FUNCTION_BLOCK FB_Stop
VAR_INPUT
(*È«¾Ö*)
	Mode:DINT;
	PowerState:DINT;
	CoupleState:DINT;
	(*GapMode*)
	GapStop:BOOL;
	(*BCGapMode*)
	BCGapStop:BOOL;
	(*SingleCarrierMode*)
	TopStop:BOOL;
	BottomStop:BOOL;
	(*TaperMode*)
	TaperStop:BOOL;
	(*DebugMode*)
	LeftTopStop:BOOL;
	RightTopStop:BOOL;
	LeftBottomStop:BOOL;
	RightBottomStop:BOOL;
END_VAR
VAR_OUTPUT
	FbID:DINT:=1001;
	GapState:DINT;
	GapBusy:BOOL;
	GapDone:BOOL;

	BCGapState:DINT;
	BCGapBusy:BOOL;
	BCGapDone:BOOL;

	TopState:DINT;
	TopBusy:BOOL;
	TopDone:BOOL;
	BottomState:DINT;
	BottomBusy:BOOL;
	BottomDone:BOOL;

	TaperState:DINT;
	TaperBusy:BOOL;
	TaperDone:BOOL;

	LeftTopState:DINT;
	LeftTopBusy:BOOL;
	LeftTopDone:BOOL;
	RightTopState:DINT;
	RightTopBusy:BOOL;
	RightTopDone:BOOL;
	LeftBottomState:DINT;
	LeftBottomBusy:BOOL;
	LeftBottomDone:BOOL;
	RightBottomState:DINT;
	RightBottomBusy:BOOL;
	RightBottomDone:BOOL;

	Error:BOOL;
	ErrorID:DINT;
END_VAR
VAR
	Top_MC_Stop: MC_Stop;
	Bottom_MC_Stop: MC_Stop;
	RightTopLin_MC_Stop: MC_Stop;
	RightBottomLin_MC_Stop: MC_Stop;
	fb_ton: TON;
	fb_ton1: TON;
	fb_ton2: TON;
	fb_ton_debug_1:TON;
	fb_ton_debug_2:TON;
	fb_ton_debug_3:TON;
	fb_ton_debug_4:TON;
	fb_ton_BC: TON;
END_VAR

IF PowerState=1 THEN
	IF Mode=1 AND CoupleState=1 THEN
		A_GapStop();
	ELSIF Mode=2 AND CoupleState=1 AND TopStop THEN
		A_TopStop();
	ELSIF Mode=2 AND CoupleState=1 AND BottomStop THEN
		A_BottomStop();
	ELSIF Mode=3 AND CoupleState=0 AND TaperStop THEN
		A_TaperStop();
	ELSIF Mode=4 AND CoupleState=0 AND LeftTopStop THEN
		A_LeftTopStop();
	ELSIF Mode=4 AND CoupleState=0 AND RightTopStop THEN
		A_RightTopStop();
	ELSIF Mode=4 AND CoupleState=0 AND LeftBottomStop THEN
		A_LeftBottomStop();
	ELSIF Mode=4 AND CoupleState=0 AND RightBottomStop THEN
		A_RightBottomStop();
	ELSIF Mode=5 AND CoupleState=0 AND BCGapStop THEN
		A_BCGapStop();
	ELSE
		FB_PlcEmergencyStop();
	END_IF
END_IF

ACTION A_BCGapStop:
IF BCGapStop THEN
BCGapBusy:=TRUE;
BCGapDone:=FALSE;
fb_ton_BC(PT:=t#100ms);
A_StopMC();
CASE BCGapState OF
	0:
		IF Top_MC_Stop.Error OR Bottom_MC_Stop.Error OR RightTopLin_MC_Stop.Error OR RightBottomLin_MC_Stop.Error THEN
			ErrorID:=1;
			BCGapState:=-100;
			Top_MC_Stop.Execute:=FALSE;
			Bottom_MC_Stop.Execute:=FALSE;
			RightTopLin_MC_Stop.Execute:=FALSE;
			RightBottomLin_MC_Stop.Execute:=FALSE;
			A_StopMC();
		ELSE
			BCGapState:=1;
		END_IF
	1:
		Top_MC_Stop.Execute:=TRUE;
		Bottom_MC_Stop.Execute:=TRUE;
		RightTopLin_MC_Stop.Execute:=TRUE;
		RightBottomLin_MC_Stop.Execute:=TRUE;
		fb_ton_BC.IN:=TRUE;
		BCGapState:=2;
	2:
		IF  NOT Top_MC_Stop.Done OR NOT Bottom_MC_Stop.Done OR NOT RightTopLin_MC_Stop.Done OR NOT RightBottomLin_MC_Stop.Done THEN
				BCGapState:=2;
		ELSE
			BCGapState:=88;
			Top_MC_Stop.Execute:=FALSE;
			Bottom_MC_Stop.Execute:=FALSE;
			RightTopLin_MC_Stop.Execute:=FALSE;
			RightBottomLin_MC_Stop.Execute:=FALSE;
			A_StopMC();
		END_IF

	88:
		BCGapStop:=FALSE;
		BCGapState:=0;
		BCGapBusy:=FALSE;
		BCGapDone:=TRUE;
		Error:=FALSE;
		ErrorID:=0;
		fb_ton_BC.IN:=FALSE;

	-100:
		FB_PlcEmergencyStop();
		BCGapStop:=FALSE;
		BCGapState:=-100;
		BCGapBusy:=FALSE;
		BCGapDone:=FALSE;
		Error:=TRUE;
		Top_MC_Stop.Execute:=FALSE;
		Bottom_MC_Stop.Execute:=FALSE;
		RightTopLin_MC_Stop.Execute:=FALSE;
		RightBottomLin_MC_Stop.Execute:=FALSE;
		A_StopMC();
		fb_ton_BC.IN:=FALSE;

END_CASE
END_IF
END_ACTION

ACTION A_BottomStop:
IF BottomStop THEN
BottomBusy:=TRUE;
BottomDone:=FALSE;
fb_ton2(PT:=t#100ms);
A_StopMC();
CASE BottomState OF
	0:
		IF Bottom_MC_Stop.Error THEN
			ErrorID:=1;
			BottomState:=-100;
			Bottom_MC_Stop.Execute:=FALSE;
			A_StopMC();
		ELSE
			BottomState:=1;
		END_IF
	1:
		Bottom_MC_Stop.Execute:=TRUE;
		fb_ton2.IN:=TRUE;
		BottomState:=2;
	2:
		IF  NOT Bottom_MC_Stop.Done THEN
				BottomState:=2;
		ELSE
			BottomState:=88;
			Bottom_MC_Stop.Execute:=FALSE;
			A_StopMC();
		END_IF

	88:
		BottomStop:=FALSE;
		BottomState:=0;
		BottomBusy:=FALSE;
		BottomDone:=TRUE;
		Error:=FALSE;
		ErrorID:=0;
		fb_ton2.IN:=FALSE;

	-100:
		FB_PlcEmergencyStop();
		BottomStop:=FALSE;
		BottomState:=-100;
		BottomBusy:=FALSE;
		BottomDone:=FALSE;
		Error:=TRUE;
		Bottom_MC_Stop.Execute:=FALSE;
		A_StopMC();
		fb_ton2.IN:=FALSE;

END_CASE
END_IF
END_ACTION

ACTION A_GapStop:
IF GapStop THEN
GapBusy:=TRUE;
GapDone:=FALSE;
fb_ton(PT:=t#100ms);
A_StopMC();
CASE GapState OF
	0:
		IF Top_MC_Stop.Error OR Bottom_MC_Stop.Error THEN
			ErrorID:=1;
			GapState:=-100;
			Top_MC_Stop.Execute:=FALSE;
			Bottom_MC_Stop.Execute:=FALSE;
			A_StopMC();
		ELSE
			GapState:=1;
		END_IF
	1:
		Top_MC_Stop.Execute:=TRUE;
		Bottom_MC_Stop.Execute:=TRUE;
		fb_ton.IN:=TRUE;
		GapState:=2;
	2:
		IF  NOT Top_MC_Stop.Done OR NOT Bottom_MC_Stop.Done THEN
				GapState:=2;
		ELSE
			GapState:=88;
			Top_MC_Stop.Execute:=FALSE;
			Bottom_MC_Stop.Execute:=FALSE;
			A_StopMC();
		END_IF

	88:
		GapStop:=FALSE;
		GapState:=0;
		GapBusy:=FALSE;
		GapDone:=TRUE;
		Error:=FALSE;
		ErrorID:=0;
		fb_ton.IN:=FALSE;

	-100:
		FB_PlcEmergencyStop();
		GapStop:=FALSE;
		GapState:=-100;
		GapBusy:=FALSE;
		GapDone:=FALSE;
		Error:=TRUE;
		Top_MC_Stop.Execute:=FALSE;
		Bottom_MC_Stop.Execute:=FALSE;
		A_StopMC();
		fb_ton.IN:=FALSE;

END_CASE
END_IF
END_ACTION

ACTION A_LeftBottomStop:
IF LeftBottomStop THEN
LeftBottomBusy:=TRUE;
LeftBottomDone:=FALSE;
fb_ton_debug_3(PT:=t#100ms);
A_StopMC();
CASE LeftBottomState OF
	0:
		IF Bottom_MC_Stop.Error THEN
			ErrorID:=41;
			LeftBottomState:=-100;
			Bottom_MC_Stop.Execute:=FALSE;
			A_StopMC();
		ELSE
			LeftBottomState:=1;
		END_IF
	1:
		Bottom_MC_Stop.Execute:=TRUE;
		fb_ton_debug_3.IN:=TRUE;
		LeftBottomState:=2;
	2:
		IF  NOT Bottom_MC_Stop.Done THEN
				LeftBottomState:=2;
		ELSE
			LeftBottomState:=88;
			Bottom_MC_Stop.Execute:=FALSE;
			A_StopMC();
		END_IF

	88:
		LeftBottomStop:=FALSE;
		LeftBottomState:=0;
		LeftBottomBusy:=FALSE;
		LeftBottomDone:=TRUE;
		Error:=FALSE;
		ErrorID:=0;
		fb_ton_debug_3.IN:=FALSE;

	-100:
		FB_PlcEmergencyStop();
		LeftBottomStop:=FALSE;
		LeftBottomState:=-100;
		LeftBottomBusy:=FALSE;
		LeftBottomDone:=FALSE;
		Error:=TRUE;
		Bottom_MC_Stop.Execute:=FALSE;
		A_StopMC();
		fb_ton_debug_3.IN:=FALSE;

END_CASE
END_IF
END_ACTION

ACTION A_LeftTopStop:
IF LeftTopStop THEN
LeftTopBusy:=TRUE;
LeftTopDone:=FALSE;
fb_ton_debug_1(PT:=t#100ms);
A_StopMC();
CASE LeftTopState OF
	0:
		IF Top_MC_Stop.Error THEN
			ErrorID:=41;
			LeftTopState:=-100;
			Top_MC_Stop.Execute:=FALSE;
			A_StopMC();
		ELSE
			LeftTopState:=1;
		END_IF
	1:
		Top_MC_Stop.Execute:=TRUE;
		fb_ton_debug_1.IN:=TRUE;
		LeftTopState:=2;
	2:
		IF  NOT Top_MC_Stop.Done THEN
				LeftTopState:=2;
		ELSE
			LeftTopState:=88;
			Top_MC_Stop.Execute:=FALSE;
			A_StopMC();
		END_IF

	88:
		LeftTopStop:=FALSE;
		LeftTopState:=0;
		LeftTopBusy:=FALSE;
		LeftTopDone:=TRUE;
		Error:=FALSE;
		ErrorID:=0;
		fb_ton_debug_1.IN:=FALSE;

	-100:
		FB_PlcEmergencyStop();
		LeftTopStop:=FALSE;
		LeftTopState:=-100;
		LeftTopBusy:=FALSE;
		LeftTopDone:=FALSE;
		Error:=TRUE;
		Top_MC_Stop.Execute:=FALSE;
		A_StopMC();
		fb_ton_debug_1.IN:=FALSE;

END_CASE
END_IF
END_ACTION

ACTION A_RightBottomStop:
IF RightBottomStop THEN
RightBottomBusy:=TRUE;
RightBottomDone:=FALSE;
fb_ton_debug_4(PT:=t#100ms);
A_StopMC();
CASE RightBottomState OF
	0:
		IF RightBottomLin_MC_Stop.Error THEN
			ErrorID:=41;
			RightBottomState:=-100;
			RightBottomLin_MC_Stop.Execute:=FALSE;
			A_StopMC();
		ELSE
			RightBottomState:=1;
		END_IF
	1:
		RightBottomLin_MC_Stop.Execute:=TRUE;
		fb_ton_debug_4.IN:=TRUE;
		RightBottomState:=2;
	2:
		IF  NOT RightBottomLin_MC_Stop.Done THEN
				RightBottomState:=2;
		ELSE
			RightBottomState:=88;
			RightBottomLin_MC_Stop.Execute:=FALSE;
			A_StopMC();
		END_IF

	88:
		RightBottomStop:=FALSE;
		RightBottomState:=0;
		RightBottomBusy:=FALSE;
		RightBottomDone:=TRUE;
		Error:=FALSE;
		ErrorID:=0;
		fb_ton_debug_4.IN:=FALSE;

	-100:
		FB_PlcEmergencyStop();
		RightBottomStop:=FALSE;
		RightBottomState:=-100;
		RightBottomBusy:=FALSE;
		RightBottomDone:=FALSE;
		Error:=TRUE;
		RightBottomLin_MC_Stop.Execute:=FALSE;
		A_StopMC();
		fb_ton_debug_4.IN:=FALSE;

END_CASE
END_IF
END_ACTION

ACTION A_RightTopStop:
IF RightTopStop THEN
RightTopBusy:=TRUE;
RightTopDone:=FALSE;
fb_ton_debug_2(PT:=t#100ms);
A_StopMC();
CASE RightTopState OF
	0:
		IF RightTopLin_MC_Stop.Error THEN
			ErrorID:=41;
			RightTopState:=-100;
			RightTopLin_MC_Stop.Execute:=FALSE;
			A_StopMC();
		ELSE
			RightTopState:=1;
		END_IF
	1:
		RightTopLin_MC_Stop.Execute:=TRUE;
		fb_ton_debug_2.IN:=TRUE;
		RightTopState:=2;
	2:
		IF  NOT RightTopLin_MC_Stop.Done THEN
				RightTopState:=2;
		ELSE
			RightTopState:=88;
			RightTopLin_MC_Stop.Execute:=FALSE;
			A_StopMC();
		END_IF

	88:
		RightTopStop:=FALSE;
		RightTopState:=0;
		RightTopBusy:=FALSE;
		RightTopDone:=TRUE;
		Error:=FALSE;
		ErrorID:=0;
		fb_ton_debug_2.IN:=FALSE;

	-100:
		FB_PlcEmergencyStop();
		RightTopStop:=FALSE;
		RightTopState:=-100;
		RightTopBusy:=FALSE;
		RightTopDone:=FALSE;
		Error:=TRUE;
		RightTopLin_MC_Stop.Execute:=FALSE;
		A_StopMC();
		fb_ton_debug_2.IN:=FALSE;

END_CASE
END_IF
END_ACTION

ACTION A_StopMC:
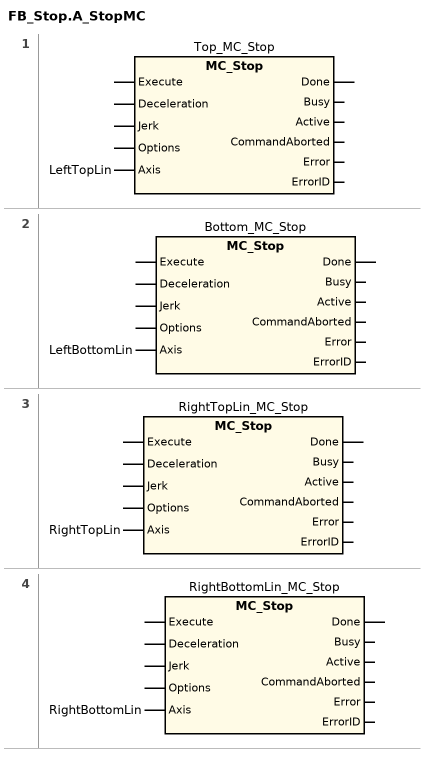
// NETWORK 1
Top_MC_Stop(Axis := LeftTopLin); // MC_Stop

// NETWORK 2
Bottom_MC_Stop(Axis := LeftBottomLin); // MC_Stop

// NETWORK 3
RightTopLin_MC_Stop(Axis := RightTopLin); // MC_Stop

// NETWORK 4
RightBottomLin_MC_Stop(Axis := RightBottomLin); // MC_Stop
END_ACTION

ACTION A_TaperStop:
IF TaperStop THEN
TaperBusy:=TRUE;
TaperDone:=FALSE;
fb_ton(PT:=t#100ms);
A_StopMC();
CASE TaperState OF
	0:
		IF RightTopLin_MC_Stop.Error  OR RightBottomLin_MC_Stop.Error THEN
			ErrorID:=1;
			TaperState:=-100;
			RightTopLin_MC_Stop.Execute:=FALSE;
			RightBottomLin_MC_Stop.Execute:=FALSE;
			A_StopMC();
		ELSE
			TaperState:=1;
		END_IF
	1:
		RightTopLin_MC_Stop.Execute:=TRUE;
		RightBottomLin_MC_Stop.Execute:=TRUE;
		fb_ton.IN:=TRUE;
		TaperState:=2;
	2:
		IF  NOT RightTopLin_MC_Stop.Done OR NOT RightBottomLin_MC_Stop.Done THEN
				TaperState:=2;
		ELSE
			TaperState:=88;
			RightTopLin_MC_Stop.Execute:=FALSE;
			RightBottomLin_MC_Stop.Execute:=FALSE;
			A_StopMC();
		END_IF

	88:
		TaperStop:=FALSE;
		TaperState:=0;
		TaperBusy:=FALSE;
		TaperDone:=TRUE;
		Error:=FALSE;
		ErrorID:=0;
		fb_ton.IN:=FALSE;

	-100:
		FB_PlcEmergencyStop();
		TaperStop:=FALSE;
		TaperState:=-100;
		TaperBusy:=FALSE;
		TaperDone:=FALSE;
		Error:=TRUE;
		RightTopLin_MC_Stop.Execute:=FALSE;
		RightBottomLin_MC_Stop.Execute:=FALSE;
		A_StopMC();
		fb_ton.IN:=FALSE;

END_CASE
END_IF
END_ACTION

ACTION A_TopStop:
IF TopStop THEN
TopBusy:=TRUE;
TopDone:=FALSE;
fb_ton1(PT:=t#100ms);
A_StopMC();
CASE TopState OF
	0:
		IF Top_MC_Stop.Error THEN
			ErrorID:=1;
			TopState:=-100;
			Top_MC_Stop.Execute:=FALSE;
			A_StopMC();
		ELSE
			TopState:=1;
		END_IF
	1:
		Top_MC_Stop.Execute:=TRUE;
		fb_ton1.IN:=TRUE;
		TopState:=2;
	2:
		IF  NOT Top_MC_Stop.Done THEN
				TopState:=2;
		ELSE
			TopState:=88;
			Top_MC_Stop.Execute:=FALSE;
			A_StopMC();
		END_IF

	88:
		TopStop:=FALSE;
		TopState:=0;
		TopBusy:=FALSE;
		TopDone:=TRUE;
		Error:=FALSE;
		ErrorID:=0;
		fb_ton1.IN:=FALSE;

	-100:
		FB_PlcEmergencyStop();
		TopStop:=FALSE;
		TopState:=-100;
		TopBusy:=FALSE;
		TopDone:=FALSE;
		Error:=TRUE;
		Top_MC_Stop.Execute:=FALSE;
		A_StopMC();
		fb_ton1.IN:=FALSE;

END_CASE
END_IF
END_ACTION

END_FUNCTION_BLOCK

(* stored: Version 1.1.0.1, ProductVersion 3.1.4024.6
   POU FB_Stop: Id {3e354bcb-4e4f-4b34-9851-51b9542d0760}, SpecialFunc None
   Action A_BCGapStop: Id {09d39807-0cc9-4816-a94c-73c13504c1f7}
   Action A_BottomStop: Id {3e5d2212-d55d-4178-a1aa-10c2e89eefb4}
   Action A_GapStop: Id {c2543639-368b-4271-b25d-0ff0da1ffa36}
   Action A_LeftBottomStop: Id {cab19fe7-18d8-423d-84e7-b2a63e643950}
   Action A_LeftTopStop: Id {2b524d72-b139-4ac0-8fb1-7a7578319dea}
   Action A_RightBottomStop: Id {e95ff139-ca76-4481-866d-edf0363d8b42}
   Action A_RightTopStop: Id {81452b6a-45dc-414d-8661-6860831ad67d}
   Action A_StopMC: Id {b171a3f0-94b4-4ac2-92c0-8ca964cc4005}
   Action A_TaperStop: Id {5bb0ea65-29f0-4cac-b793-f3368de82a9d}
   Action A_TopStop: Id {35574051-d064-41d9-8c90-d1d9b62d4922} *)
